// This interface defines the behaviour of a stopwatch, a type of timing source 
// used to measure the elapsed time between the start and stop actions. It can
// be cleared to reset the elapsed time and is useful for timing events,
// measuring durations, or performance monitoring.
INTERFACE I_Stopwatch EXTENDS I_TimingSource

// Clears the stopwatch, resetting the elapsed time to zero.
METHOD Clear
VAR_INPUT
END_VAR
END_METHOD

// The elapsed time measured by the stopwatch since it was started.
// [get] Returns the elapsed time.
PROPERTY ElapsedTime  : LTIME
GET
END_GET
END_PROPERTY

// Indicates whether the stopwatch is currently running.
// [get] Returns TRUE if the stopwatch is running; otherwise, FALSE.
PROPERTY IsRunning  : BOOL
GET
END_GET
END_PROPERTY

// Starts the stopwatch, beginning the measurement of elapsed time.
METHOD Start
VAR_INPUT
END_VAR
END_METHOD

// Stops the stopwatch, halting the measurement of elapsed time.
METHOD Stop
VAR_INPUT
END_VAR
END_METHOD

END_INTERFACE

(* stored: Version 1.1.0.1
   Itf I_Stopwatch: Id {929dffcf-71a3-4efe-adf8-2dcc46c84bab}
   Method Clear: Id {d22b2e11-2c0f-459b-828c-b430a30d9346}
   Property ElapsedTime: Id {58223e66-6c8f-4dc4-a262-2221f74c1c4d}
   Get Get: Id {6c02b00e-aedc-49fd-997f-c22f8c3378e4}
   Property IsRunning: Id {7c2b704e-7364-47dc-a532-fe111f9a98a0}
   Get Get: Id {43c50cf2-1b24-4139-b1fe-dd7fc8179ce1}
   Method Start: Id {ade4cee3-7161-488b-ad4b-d79881acbdec}
   Method Stop: Id {fc64b532-35a4-43ff-95c0-43f64680b17b} *)
